// TIA Portal V17 export
// export: Created 2025-03-10T13:11:52.5932602Z, ExportSetting WithDefaults, DisplayName Totally Integrated Automation Portal, DisplayVersion V17 Update 8, DisplayName TIA Portal Openness, DisplayVersion V17 Update 8, DisplayName TIA Portal Version Control Interface, DisplayVersion V17, DisplayName SINAMICS Startdrive Advanced, DisplayVersion V17 SP2, DisplayName SINAMICS Startdrive G110M, G120, G120C, G120D, G120P, G115D, DisplayVersion V17 SP2, DisplayName SINAMICS Startdrive G130, G150, S120, S150, SINAMICS MV, S210, DisplayVersion V17 SP2, DisplayName STEP 7 Professional, DisplayVersion V17 Update 8, DisplayName SINUMERIK ONE STEP 7 Toolbox, DisplayVersion V17 Update 12, DisplayName SINUMERIK 840D sl STEP 7 Toolbox, DisplayVersion V17 Update 12, DisplayName STEP 7 Safety, DisplayVersion V17 Update 6, DisplayName WinCC Advanced, DisplayVersion V17 Update 8
TYPE "LBP_typeAlarmMsgs"
TITLE = PLC-Error / Messages / PLC errores/avisos / PLC-Fehler / Meldungen
// User data type for block LBP_AlarmMessage [DB2] / Tipo de dato de usuario para bloque LBP_AlarmMessage [DB2] / Anwender-Datentyp für Baustein LBP_AlarmMessage [DB2]
// stored: IsFailsafeCompliant false
   STRUCT
      Chan : Array[1..10] of Struct   // Von Kanal 1..10 / From Channel 1..10 / Desde el canal 1..10
         FDD : Array[0..15] of Bool;   // Vorschub deaktivieren / Feed disable / Desactivar avance
         RID : Array[0..15] of Bool;   // Einlesen deaktivieren / Read-in disable / Desactivar lectura
         NCSD : Array[0..15] of Bool;   // NC Start deaktivieren / NC start disable / Desactivar Marcha CN
         FdStop_1 : Array[0..15] of Bool;   // Vorschub-Stopp GEO-Achse 1 / Feed stop GEOaxis 1 / Parada del avance eje geométrico 1
         FdStop_2 : Array[0..15] of Bool;   // Vorschub-Stopp GEO-Achse 2 / Feed stop GEOaxis 2 / Parada del avance eje geométrico 2
         FdStop_3 : Array[0..15] of Bool;   // Vorschub-Stopp GEO-Achse 3 / Feed stop GEOaxis 3 / Parada del avance eje geométrico 3
      END_STRUCT;
      Axis : Array[1..31] of Struct   // Von Achse 1..31 / From Axis 1..31 / Desde el eje 1..31
         FdStop : Array[0..15] of Bool;   // Vorschub-Stopp Achse/Spindel / Feed stop axis/spindle / Parada del avance eje/cabezal
      END_STRUCT;
      AddValUserA0 : Array[0..63] of Int;   // Zusätzlicher Wert für Alarme im Anwenderbereich 0 (700000..700063) / Additional value for alarms in the user area 0 (700000..700063) / Valor adicional para alarmas en el área de usuario 0 (700000..700063)
      ChanA : Array[1..10] of Struct   // Von Kanal 1..10 / From Channel 1..10 / Desde el canal 1..10
         FDD_5C00xx : Array[0..15] of Bool;   // Vorschub deaktivieren Alarm Nr. 5C0000..5C0015 / Feed disable Alarm no. 5C0000..5C0015 / Desactivar avance n.º alarma 5C0000..5C0015
         FDD_RID_5C01xx : Array[0..31] of Bool;   // Vorschub und Einlesen deaktivieren Alarm Nr. 5C0100..5C0131 / Feed and read-in disable Alarm no. 5C0100..5C0131 / Desactivar avance y lectura n.º alarma 5C0100..5C0131
         RID_5C02xx : Array[0..31] of Bool;   // Einlesen deaktivieren Alarm Nr. 5C0200..5C0231 / Read-in disable Alarm no. 5C0200..5C0231 / Desactivar lectura n.º alarma 5C0200..5C0231
         NCSD_5C03xx : Array[0..15] of Bool;   // NC Start deaktivieren Alarm Nr. 5C0300..5C0315 / NC start disable Alarm no. 5C0300..5C0315 / Desactivar Marcha CN n.º alarma 5C0300..5C0315
         FdStop_1_5C11xx : Array[0..15] of Bool;   // Vorschub-Stopp GEO-Achse 1 Alarm Nr. 5C1100..5C1115 / Feed stop GEOaxis 1 Alarm no. 5C1100..5C1115 / Parada de avance eje geométrico 1 n.º alarma 5C1100..5C1115
         FdStop_2_5C12xx : Array[0..15] of Bool;   // Vorschub-Stopp GEO-Achse 2 Alarm Nr. 5C1200..5C1215 / Feed stop GEOaxis 2 Alarm no. 5C1200..5C1215 / Parada de avance eje geométrico 2 n.º alarma 5C1200..5C1215
         FdStop_3_5C13xx : Array[0..15] of Bool;   // Vorschub-Stopp GEO-Achse 3 Alarm Nr. 5C1300..5C1315 / Feed stop GEOaxis 3 Alarm no. 5C1300..5C1315 / Parada de avance eje geométrico 3 n.º alarma 5C1300..5C1315
      END_STRUCT;
      AxisA : Array[1..31] of Struct   // Von Achse 1..31 / From Axis 1..31 / Desde el eje 1..31
         AAFdStop60AAxx : Array[0..15] of Bool;   // Vorschub-Stopp Achse/Spindel / Feed stop axis/spindle / Parada del avance eje/cabezal
      END_STRUCT;
      res552 : Word;   // Reserviert / Reserved / Reservado
      UserA : Array[0..63] of Struct
         A70UUxx : Array[0..63] of Bool;   // Alarm 70UU00..70UU63 (Anwender-Bereich) / Alarm 70UU00..70UU63 (user area) / Alarma 70UU00..70UU63 (área de usuario)
      END_STRUCT;
   END_STRUCT;
   // // Chan[2].FDD : Vorschub deaktivieren / Feed disable / Desactivar avance
   // // Chan[3].FDD : Vorschub deaktivieren / Feed disable / Desactivar avance
   // // Chan[4].FDD : Vorschub deaktivieren / Feed disable / Desactivar avance
   // // Chan[5].FDD : Vorschub deaktivieren / Feed disable / Desactivar avance
   // // Chan[6].FDD : Vorschub deaktivieren / Feed disable / Desactivar avance
   // // Chan[7].FDD : Vorschub deaktivieren / Feed disable / Desactivar avance
   // // Chan[8].FDD : Vorschub deaktivieren / Feed disable / Desactivar avance
   // // Chan[9].FDD : Vorschub deaktivieren / Feed disable / Desactivar avance
   // // Chan[10].FDD : Vorschub deaktivieren / Feed disable / Desactivar avance
   // // Chan[2].RID : Einlesen deaktivieren / Read-in disable / Desactivar lectura
   // // Chan[3].RID : Einlesen deaktivieren / Read-in disable / Desactivar lectura
   // // Chan[4].RID : Einlesen deaktivieren / Read-in disable / Desactivar lectura
   // // Chan[5].RID : Einlesen deaktivieren / Read-in disable / Desactivar lectura
   // // Chan[6].RID : Einlesen deaktivieren / Read-in disable / Desactivar lectura
   // // Chan[7].RID : Einlesen deaktivieren / Read-in disable / Desactivar lectura
   // // Chan[8].RID : Einlesen deaktivieren / Read-in disable / Desactivar lectura
   // // Chan[9].RID : Einlesen deaktivieren / Read-in disable / Desactivar lectura
   // // Chan[10].RID : Einlesen deaktivieren / Read-in disable / Desactivar lectura
   // // Chan[2].NCSD : NC Start deaktivieren / NC start disable / Desactivar Marcha CN
   // // Chan[3].NCSD : NC Start deaktivieren / NC start disable / Desactivar Marcha CN
   // // Chan[4].NCSD : NC Start deaktivieren / NC start disable / Desactivar Marcha CN
   // // Chan[5].NCSD : NC Start deaktivieren / NC start disable / Desactivar Marcha CN
   // // Chan[6].NCSD : NC Start deaktivieren / NC start disable / Desactivar Marcha CN
   // // Chan[7].NCSD : NC Start deaktivieren / NC start disable / Desactivar Marcha CN
   // // Chan[8].NCSD : NC Start deaktivieren / NC start disable / Desactivar Marcha CN
   // // Chan[9].NCSD : NC Start deaktivieren / NC start disable / Desactivar Marcha CN
   // // Chan[10].NCSD : NC Start deaktivieren / NC start disable / Desactivar Marcha CN
   // // Chan[2].FdStop_1 : Vorschub-Stopp GEO-Achse 1 / Feed stop GEOaxis 1 / Parada del avance eje geométrico 1
   // // Chan[3].FdStop_1 : Vorschub-Stopp GEO-Achse 1 / Feed stop GEOaxis 1 / Parada del avance eje geométrico 1
   // // Chan[4].FdStop_1 : Vorschub-Stopp GEO-Achse 1 / Feed stop GEOaxis 1 / Parada del avance eje geométrico 1
   // // Chan[5].FdStop_1 : Vorschub-Stopp GEO-Achse 1 / Feed stop GEOaxis 1 / Parada del avance eje geométrico 1
   // // Chan[6].FdStop_1 : Vorschub-Stopp GEO-Achse 1 / Feed stop GEOaxis 1 / Parada del avance eje geométrico 1
   // // Chan[7].FdStop_1 : Vorschub-Stopp GEO-Achse 1 / Feed stop GEOaxis 1 / Parada del avance eje geométrico 1
   // // Chan[8].FdStop_1 : Vorschub-Stopp GEO-Achse 1 / Feed stop GEOaxis 1 / Parada del avance eje geométrico 1
   // // Chan[9].FdStop_1 : Vorschub-Stopp GEO-Achse 1 / Feed stop GEOaxis 1 / Parada del avance eje geométrico 1
   // // Chan[10].FdStop_1 : Vorschub-Stopp GEO-Achse 1 / Feed stop GEOaxis 1 / Parada del avance eje geométrico 1
   // // Chan[2].FdStop_2 : Vorschub-Stopp GEO-Achse 2 / Feed stop GEOaxis 2 / Parada del avance eje geométrico 2
   // // Chan[3].FdStop_2 : Vorschub-Stopp GEO-Achse 2 / Feed stop GEOaxis 2 / Parada del avance eje geométrico 2
   // // Chan[4].FdStop_2 : Vorschub-Stopp GEO-Achse 2 / Feed stop GEOaxis 2 / Parada del avance eje geométrico 2
   // // Chan[5].FdStop_2 : Vorschub-Stopp GEO-Achse 2 / Feed stop GEOaxis 2 / Parada del avance eje geométrico 2
   // // Chan[6].FdStop_2 : Vorschub-Stopp GEO-Achse 2 / Feed stop GEOaxis 2 / Parada del avance eje geométrico 2
   // // Chan[7].FdStop_2 : Vorschub-Stopp GEO-Achse 2 / Feed stop GEOaxis 2 / Parada del avance eje geométrico 2
   // // Chan[8].FdStop_2 : Vorschub-Stopp GEO-Achse 2 / Feed stop GEOaxis 2 / Parada del avance eje geométrico 2
   // // Chan[9].FdStop_2 : Vorschub-Stopp GEO-Achse 2 / Feed stop GEOaxis 2 / Parada del avance eje geométrico 2
   // // Chan[10].FdStop_2 : Vorschub-Stopp GEO-Achse 2 / Feed stop GEOaxis 2 / Parada del avance eje geométrico 2
   // // Chan[2].FdStop_3 : Vorschub-Stopp GEO-Achse 3 / Feed stop GEOaxis 3 / Parada del avance eje geométrico 3
   // // Chan[3].FdStop_3 : Vorschub-Stopp GEO-Achse 3 / Feed stop GEOaxis 3 / Parada del avance eje geométrico 3
   // // Chan[4].FdStop_3 : Vorschub-Stopp GEO-Achse 3 / Feed stop GEOaxis 3 / Parada del avance eje geométrico 3
   // // Chan[5].FdStop_3 : Vorschub-Stopp GEO-Achse 3 / Feed stop GEOaxis 3 / Parada del avance eje geométrico 3
   // // Chan[6].FdStop_3 : Vorschub-Stopp GEO-Achse 3 / Feed stop GEOaxis 3 / Parada del avance eje geométrico 3
   // // Chan[7].FdStop_3 : Vorschub-Stopp GEO-Achse 3 / Feed stop GEOaxis 3 / Parada del avance eje geométrico 3
   // // Chan[8].FdStop_3 : Vorschub-Stopp GEO-Achse 3 / Feed stop GEOaxis 3 / Parada del avance eje geométrico 3
   // // Chan[9].FdStop_3 : Vorschub-Stopp GEO-Achse 3 / Feed stop GEOaxis 3 / Parada del avance eje geométrico 3
   // // Chan[10].FdStop_3 : Vorschub-Stopp GEO-Achse 3 / Feed stop GEOaxis 3 / Parada del avance eje geométrico 3
   // // Chan[1] : Von Kanal 1..10 / From Channel 1..10 / Desde el canal 1..10
   // // Chan[2] : Von Kanal 1..10 / From Channel 1..10 / Desde el canal 1..10
   // // Chan[3] : Von Kanal 1..10 / From Channel 1..10 / Desde el canal 1..10
   // // Chan[4] : Von Kanal 1..10 / From Channel 1..10 / Desde el canal 1..10
   // // Chan[5] : Von Kanal 1..10 / From Channel 1..10 / Desde el canal 1..10
   // // Chan[6] : Von Kanal 1..10 / From Channel 1..10 / Desde el canal 1..10
   // // Chan[7] : Von Kanal 1..10 / From Channel 1..10 / Desde el canal 1..10
   // // Chan[8] : Von Kanal 1..10 / From Channel 1..10 / Desde el canal 1..10
   // // Chan[9] : Von Kanal 1..10 / From Channel 1..10 / Desde el canal 1..10
   // // Chan[10] : Von Kanal 1..10 / From Channel 1..10 / Desde el canal 1..10
   // // Axis[2].FdStop : Vorschub-Stopp Achse/Spindel / Feed stop axis/spindle / Parada del avance eje/cabezal
   // // Axis[3].FdStop : Vorschub-Stopp Achse/Spindel / Feed stop axis/spindle / Parada del avance eje/cabezal
   // // Axis[4].FdStop : Vorschub-Stopp Achse/Spindel / Feed stop axis/spindle / Parada del avance eje/cabezal
   // // Axis[5].FdStop : Vorschub-Stopp Achse/Spindel / Feed stop axis/spindle / Parada del avance eje/cabezal
   // // Axis[6].FdStop : Vorschub-Stopp Achse/Spindel / Feed stop axis/spindle / Parada del avance eje/cabezal
   // // Axis[7].FdStop : Vorschub-Stopp Achse/Spindel / Feed stop axis/spindle / Parada del avance eje/cabezal
   // // Axis[8].FdStop : Vorschub-Stopp Achse/Spindel / Feed stop axis/spindle / Parada del avance eje/cabezal
   // // Axis[9].FdStop : Vorschub-Stopp Achse/Spindel / Feed stop axis/spindle / Parada del avance eje/cabezal
   // // Axis[10].FdStop : Vorschub-Stopp Achse/Spindel / Feed stop axis/spindle / Parada del avance eje/cabezal
   // // Axis[11].FdStop : Vorschub-Stopp Achse/Spindel / Feed stop axis/spindle / Parada del avance eje/cabezal
   // // Axis[12].FdStop : Vorschub-Stopp Achse/Spindel / Feed stop axis/spindle / Parada del avance eje/cabezal
   // // Axis[13].FdStop : Vorschub-Stopp Achse/Spindel / Feed stop axis/spindle / Parada del avance eje/cabezal
   // // Axis[14].FdStop : Vorschub-Stopp Achse/Spindel / Feed stop axis/spindle / Parada del avance eje/cabezal
   // // Axis[15].FdStop : Vorschub-Stopp Achse/Spindel / Feed stop axis/spindle / Parada del avance eje/cabezal
   // // Axis[16].FdStop : Vorschub-Stopp Achse/Spindel / Feed stop axis/spindle / Parada del avance eje/cabezal
   // // Axis[17].FdStop : Vorschub-Stopp Achse/Spindel / Feed stop axis/spindle / Parada del avance eje/cabezal
   // // Axis[18].FdStop : Vorschub-Stopp Achse/Spindel / Feed stop axis/spindle / Parada del avance eje/cabezal
   // // Axis[19].FdStop : Vorschub-Stopp Achse/Spindel / Feed stop axis/spindle / Parada del avance eje/cabezal
   // // Axis[20].FdStop : Vorschub-Stopp Achse/Spindel / Feed stop axis/spindle / Parada del avance eje/cabezal
   // // Axis[21].FdStop : Vorschub-Stopp Achse/Spindel / Feed stop axis/spindle / Parada del avance eje/cabezal
   // // Axis[22].FdStop : Vorschub-Stopp Achse/Spindel / Feed stop axis/spindle / Parada del avance eje/cabezal
   // // Axis[23].FdStop : Vorschub-Stopp Achse/Spindel / Feed stop axis/spindle / Parada del avance eje/cabezal
   // // Axis[24].FdStop : Vorschub-Stopp Achse/Spindel / Feed stop axis/spindle / Parada del avance eje/cabezal
   // // Axis[25].FdStop : Vorschub-Stopp Achse/Spindel / Feed stop axis/spindle / Parada del avance eje/cabezal
   // // Axis[26].FdStop : Vorschub-Stopp Achse/Spindel / Feed stop axis/spindle / Parada del avance eje/cabezal
   // // Axis[27].FdStop : Vorschub-Stopp Achse/Spindel / Feed stop axis/spindle / Parada del avance eje/cabezal
   // // Axis[28].FdStop : Vorschub-Stopp Achse/Spindel / Feed stop axis/spindle / Parada del avance eje/cabezal
   // // Axis[29].FdStop : Vorschub-Stopp Achse/Spindel / Feed stop axis/spindle / Parada del avance eje/cabezal
   // // Axis[30].FdStop : Vorschub-Stopp Achse/Spindel / Feed stop axis/spindle / Parada del avance eje/cabezal
   // // Axis[31].FdStop : Vorschub-Stopp Achse/Spindel / Feed stop axis/spindle / Parada del avance eje/cabezal
   // // Axis[1] : Von Achse 1..31 / From Axis 1..31 / Desde el eje 1..31
   // // Axis[2] : Von Achse 1..31 / From Axis 1..31 / Desde el eje 1..31
   // // Axis[3] : Von Achse 1..31 / From Axis 1..31 / Desde el eje 1..31
   // // Axis[4] : Von Achse 1..31 / From Axis 1..31 / Desde el eje 1..31
   // // Axis[5] : Von Achse 1..31 / From Axis 1..31 / Desde el eje 1..31
   // // Axis[6] : Von Achse 1..31 / From Axis 1..31 / Desde el eje 1..31
   // // Axis[7] : Von Achse 1..31 / From Axis 1..31 / Desde el eje 1..31
   // // Axis[8] : Von Achse 1..31 / From Axis 1..31 / Desde el eje 1..31
   // // Axis[9] : Von Achse 1..31 / From Axis 1..31 / Desde el eje 1..31
   // // Axis[10] : Von Achse 1..31 / From Axis 1..31 / Desde el eje 1..31
   // // Axis[11] : Von Achse 1..31 / From Axis 1..31 / Desde el eje 1..31
   // // Axis[12] : Von Achse 1..31 / From Axis 1..31 / Desde el eje 1..31
   // // Axis[13] : Von Achse 1..31 / From Axis 1..31 / Desde el eje 1..31
   // // Axis[14] : Von Achse 1..31 / From Axis 1..31 / Desde el eje 1..31
   // // Axis[15] : Von Achse 1..31 / From Axis 1..31 / Desde el eje 1..31
   // // Axis[16] : Von Achse 1..31 / From Axis 1..31 / Desde el eje 1..31
   // // Axis[17] : Von Achse 1..31 / From Axis 1..31 / Desde el eje 1..31
   // // Axis[18] : Von Achse 1..31 / From Axis 1..31 / Desde el eje 1..31
   // // Axis[19] : Von Achse 1..31 / From Axis 1..31 / Desde el eje 1..31
   // // Axis[20] : Von Achse 1..31 / From Axis 1..31 / Desde el eje 1..31
   // // Axis[21] : Von Achse 1..31 / From Axis 1..31 / Desde el eje 1..31
   // // Axis[22] : Von Achse 1..31 / From Axis 1..31 / Desde el eje 1..31
   // // Axis[23] : Von Achse 1..31 / From Axis 1..31 / Desde el eje 1..31
   // // Axis[24] : Von Achse 1..31 / From Axis 1..31 / Desde el eje 1..31
   // // Axis[25] : Von Achse 1..31 / From Axis 1..31 / Desde el eje 1..31
   // // Axis[26] : Von Achse 1..31 / From Axis 1..31 / Desde el eje 1..31
   // // Axis[27] : Von Achse 1..31 / From Axis 1..31 / Desde el eje 1..31
   // // Axis[28] : Von Achse 1..31 / From Axis 1..31 / Desde el eje 1..31
   // // Axis[29] : Von Achse 1..31 / From Axis 1..31 / Desde el eje 1..31
   // // Axis[30] : Von Achse 1..31 / From Axis 1..31 / Desde el eje 1..31
   // // Axis[31] : Von Achse 1..31 / From Axis 1..31 / Desde el eje 1..31
   // // ChanA[2].FDD_5C00xx : Vorschub deaktivieren Alarm Nr. 5C0000..5C0015 / Feed disable Alarm no. 5C0000..5C0015 / Desactivar avance n.º alarma 5C0000..5C0015
   // // ChanA[3].FDD_5C00xx : Vorschub deaktivieren Alarm Nr. 5C0000..5C0015 / Feed disable Alarm no. 5C0000..5C0015 / Desactivar avance n.º alarma 5C0000..5C0015
   // // ChanA[4].FDD_5C00xx : Vorschub deaktivieren Alarm Nr. 5C0000..5C0015 / Feed disable Alarm no. 5C0000..5C0015 / Desactivar avance n.º alarma 5C0000..5C0015
   // // ChanA[5].FDD_5C00xx : Vorschub deaktivieren Alarm Nr. 5C0000..5C0015 / Feed disable Alarm no. 5C0000..5C0015 / Desactivar avance n.º alarma 5C0000..5C0015
   // // ChanA[6].FDD_5C00xx : Vorschub deaktivieren Alarm Nr. 5C0000..5C0015 / Feed disable Alarm no. 5C0000..5C0015 / Desactivar avance n.º alarma 5C0000..5C0015
   // // ChanA[7].FDD_5C00xx : Vorschub deaktivieren Alarm Nr. 5C0000..5C0015 / Feed disable Alarm no. 5C0000..5C0015 / Desactivar avance n.º alarma 5C0000..5C0015
   // // ChanA[8].FDD_5C00xx : Vorschub deaktivieren Alarm Nr. 5C0000..5C0015 / Feed disable Alarm no. 5C0000..5C0015 / Desactivar avance n.º alarma 5C0000..5C0015
   // // ChanA[9].FDD_5C00xx : Vorschub deaktivieren Alarm Nr. 5C0000..5C0015 / Feed disable Alarm no. 5C0000..5C0015 / Desactivar avance n.º alarma 5C0000..5C0015
   // // ChanA[10].FDD_5C00xx : Vorschub deaktivieren Alarm Nr. 5C0000..5C0015 / Feed disable Alarm no. 5C0000..5C0015 / Desactivar avance n.º alarma 5C0000..5C0015
   // // ChanA[2].FDD_RID_5C01xx : Vorschub und Einlesen deaktivieren Alarm Nr. 5C0100..5C0131 / Feed and read-in disable Alarm no. 5C0100..5C0131 / Desactivar avance y lectura n.º alarma 5C0100..5C0131
   // // ChanA[3].FDD_RID_5C01xx : Vorschub und Einlesen deaktivieren Alarm Nr. 5C0100..5C0131 / Feed and read-in disable Alarm no. 5C0100..5C0131 / Desactivar avance y lectura n.º alarma 5C0100..5C0131
   // // ChanA[4].FDD_RID_5C01xx : Vorschub und Einlesen deaktivieren Alarm Nr. 5C0100..5C0131 / Feed and read-in disable Alarm no. 5C0100..5C0131 / Desactivar avance y lectura n.º alarma 5C0100..5C0131
   // // ChanA[5].FDD_RID_5C01xx : Vorschub und Einlesen deaktivieren Alarm Nr. 5C0100..5C0131 / Feed and read-in disable Alarm no. 5C0100..5C0131 / Desactivar avance y lectura n.º alarma 5C0100..5C0131
   // // ChanA[6].FDD_RID_5C01xx : Vorschub und Einlesen deaktivieren Alarm Nr. 5C0100..5C0131 / Feed and read-in disable Alarm no. 5C0100..5C0131 / Desactivar avance y lectura n.º alarma 5C0100..5C0131
   // // ChanA[7].FDD_RID_5C01xx : Vorschub und Einlesen deaktivieren Alarm Nr. 5C0100..5C0131 / Feed and read-in disable Alarm no. 5C0100..5C0131 / Desactivar avance y lectura n.º alarma 5C0100..5C0131
   // // ChanA[8].FDD_RID_5C01xx : Vorschub und Einlesen deaktivieren Alarm Nr. 5C0100..5C0131 / Feed and read-in disable Alarm no. 5C0100..5C0131 / Desactivar avance y lectura n.º alarma 5C0100..5C0131
   // // ChanA[9].FDD_RID_5C01xx : Vorschub und Einlesen deaktivieren Alarm Nr. 5C0100..5C0131 / Feed and read-in disable Alarm no. 5C0100..5C0131 / Desactivar avance y lectura n.º alarma 5C0100..5C0131
   // // ChanA[10].FDD_RID_5C01xx : Vorschub und Einlesen deaktivieren Alarm Nr. 5C0100..5C0131 / Feed and read-in disable Alarm no. 5C0100..5C0131 / Desactivar avance y lectura n.º alarma 5C0100..5C0131
   // // ChanA[2].RID_5C02xx : Einlesen deaktivieren Alarm Nr. 5C0200..5C0231 / Read-in disable Alarm no. 5C0200..5C0231 / Desactivar lectura n.º alarma 5C0200..5C0231
   // // ChanA[3].RID_5C02xx : Einlesen deaktivieren Alarm Nr. 5C0200..5C0231 / Read-in disable Alarm no. 5C0200..5C0231 / Desactivar lectura n.º alarma 5C0200..5C0231
   // // ChanA[4].RID_5C02xx : Einlesen deaktivieren Alarm Nr. 5C0200..5C0231 / Read-in disable Alarm no. 5C0200..5C0231 / Desactivar lectura n.º alarma 5C0200..5C0231
   // // ChanA[5].RID_5C02xx : Einlesen deaktivieren Alarm Nr. 5C0200..5C0231 / Read-in disable Alarm no. 5C0200..5C0231 / Desactivar lectura n.º alarma 5C0200..5C0231
   // // ChanA[6].RID_5C02xx : Einlesen deaktivieren Alarm Nr. 5C0200..5C0231 / Read-in disable Alarm no. 5C0200..5C0231 / Desactivar lectura n.º alarma 5C0200..5C0231
   // // ChanA[7].RID_5C02xx : Einlesen deaktivieren Alarm Nr. 5C0200..5C0231 / Read-in disable Alarm no. 5C0200..5C0231 / Desactivar lectura n.º alarma 5C0200..5C0231
   // // ChanA[8].RID_5C02xx : Einlesen deaktivieren Alarm Nr. 5C0200..5C0231 / Read-in disable Alarm no. 5C0200..5C0231 / Desactivar lectura n.º alarma 5C0200..5C0231
   // // ChanA[9].RID_5C02xx : Einlesen deaktivieren Alarm Nr. 5C0200..5C0231 / Read-in disable Alarm no. 5C0200..5C0231 / Desactivar lectura n.º alarma 5C0200..5C0231
   // // ChanA[10].RID_5C02xx : Einlesen deaktivieren Alarm Nr. 5C0200..5C0231 / Read-in disable Alarm no. 5C0200..5C0231 / Desactivar lectura n.º alarma 5C0200..5C0231
   // // ChanA[2].NCSD_5C03xx : NC Start deaktivieren Alarm Nr. 5C0300..5C0315 / NC start disable Alarm no. 5C0300..5C0315 / Desactivar Marcha CN n.º alarma 5C0300..5C0315
   // // ChanA[3].NCSD_5C03xx : NC Start deaktivieren Alarm Nr. 5C0300..5C0315 / NC start disable Alarm no. 5C0300..5C0315 / Desactivar Marcha CN n.º alarma 5C0300..5C0315
   // // ChanA[4].NCSD_5C03xx : NC Start deaktivieren Alarm Nr. 5C0300..5C0315 / NC start disable Alarm no. 5C0300..5C0315 / Desactivar Marcha CN n.º alarma 5C0300..5C0315
   // // ChanA[5].NCSD_5C03xx : NC Start deaktivieren Alarm Nr. 5C0300..5C0315 / NC start disable Alarm no. 5C0300..5C0315 / Desactivar Marcha CN n.º alarma 5C0300..5C0315
   // // ChanA[6].NCSD_5C03xx : NC Start deaktivieren Alarm Nr. 5C0300..5C0315 / NC start disable Alarm no. 5C0300..5C0315 / Desactivar Marcha CN n.º alarma 5C0300..5C0315
   // // ChanA[7].NCSD_5C03xx : NC Start deaktivieren Alarm Nr. 5C0300..5C0315 / NC start disable Alarm no. 5C0300..5C0315 / Desactivar Marcha CN n.º alarma 5C0300..5C0315
   // // ChanA[8].NCSD_5C03xx : NC Start deaktivieren Alarm Nr. 5C0300..5C0315 / NC start disable Alarm no. 5C0300..5C0315 / Desactivar Marcha CN n.º alarma 5C0300..5C0315
   // // ChanA[9].NCSD_5C03xx : NC Start deaktivieren Alarm Nr. 5C0300..5C0315 / NC start disable Alarm no. 5C0300..5C0315 / Desactivar Marcha CN n.º alarma 5C0300..5C0315
   // // ChanA[10].NCSD_5C03xx : NC Start deaktivieren Alarm Nr. 5C0300..5C0315 / NC start disable Alarm no. 5C0300..5C0315 / Desactivar Marcha CN n.º alarma 5C0300..5C0315
   // // ChanA[2].FdStop_1_5C11xx : Vorschub-Stopp GEO-Achse 1 Alarm Nr. 5C1100..5C1115 / Feed stop GEOaxis 1 Alarm no. 5C1100..5C1115 / Parada de avance eje geométrico 1 n.º alarma 5C1100..5C1115
   // // ChanA[3].FdStop_1_5C11xx : Vorschub-Stopp GEO-Achse 1 Alarm Nr. 5C1100..5C1115 / Feed stop GEOaxis 1 Alarm no. 5C1100..5C1115 / Parada de avance eje geométrico 1 n.º alarma 5C1100..5C1115
   // // ChanA[4].FdStop_1_5C11xx : Vorschub-Stopp GEO-Achse 1 Alarm Nr. 5C1100..5C1115 / Feed stop GEOaxis 1 Alarm no. 5C1100..5C1115 / Parada de avance eje geométrico 1 n.º alarma 5C1100..5C1115
   // // ChanA[5].FdStop_1_5C11xx : Vorschub-Stopp GEO-Achse 1 Alarm Nr. 5C1100..5C1115 / Feed stop GEOaxis 1 Alarm no. 5C1100..5C1115 / Parada de avance eje geométrico 1 n.º alarma 5C1100..5C1115
   // // ChanA[6].FdStop_1_5C11xx : Vorschub-Stopp GEO-Achse 1 Alarm Nr. 5C1100..5C1115 / Feed stop GEOaxis 1 Alarm no. 5C1100..5C1115 / Parada de avance eje geométrico 1 n.º alarma 5C1100..5C1115
   // // ChanA[7].FdStop_1_5C11xx : Vorschub-Stopp GEO-Achse 1 Alarm Nr. 5C1100..5C1115 / Feed stop GEOaxis 1 Alarm no. 5C1100..5C1115 / Parada de avance eje geométrico 1 n.º alarma 5C1100..5C1115
   // // ChanA[8].FdStop_1_5C11xx : Vorschub-Stopp GEO-Achse 1 Alarm Nr. 5C1100..5C1115 / Feed stop GEOaxis 1 Alarm no. 5C1100..5C1115 / Parada de avance eje geométrico 1 n.º alarma 5C1100..5C1115
   // // ChanA[9].FdStop_1_5C11xx : Vorschub-Stopp GEO-Achse 1 Alarm Nr. 5C1100..5C1115 / Feed stop GEOaxis 1 Alarm no. 5C1100..5C1115 / Parada de avance eje geométrico 1 n.º alarma 5C1100..5C1115
   // // ChanA[10].FdStop_1_5C11xx : Vorschub-Stopp GEO-Achse 1 Alarm Nr. 5C1100..5C1115 / Feed stop GEOaxis 1 Alarm no. 5C1100..5C1115 / Parada de avance eje geométrico 1 n.º alarma 5C1100..5C1115
   // // ChanA[2].FdStop_2_5C12xx : Vorschub-Stopp GEO-Achse 2 Alarm Nr. 5C1200..5C1215 / Feed stop GEOaxis 2 Alarm no. 5C1200..5C1215 / Parada de avance eje geométrico 2 n.º alarma 5C1200..5C1215
   // // ChanA[3].FdStop_2_5C12xx : Vorschub-Stopp GEO-Achse 2 Alarm Nr. 5C1200..5C1215 / Feed stop GEOaxis 2 Alarm no. 5C1200..5C1215 / Parada de avance eje geométrico 2 n.º alarma 5C1200..5C1215
   // // ChanA[4].FdStop_2_5C12xx : Vorschub-Stopp GEO-Achse 2 Alarm Nr. 5C1200..5C1215 / Feed stop GEOaxis 2 Alarm no. 5C1200..5C1215 / Parada de avance eje geométrico 2 n.º alarma 5C1200..5C1215
   // // ChanA[5].FdStop_2_5C12xx : Vorschub-Stopp GEO-Achse 2 Alarm Nr. 5C1200..5C1215 / Feed stop GEOaxis 2 Alarm no. 5C1200..5C1215 / Parada de avance eje geométrico 2 n.º alarma 5C1200..5C1215
   // // ChanA[6].FdStop_2_5C12xx : Vorschub-Stopp GEO-Achse 2 Alarm Nr. 5C1200..5C1215 / Feed stop GEOaxis 2 Alarm no. 5C1200..5C1215 / Parada de avance eje geométrico 2 n.º alarma 5C1200..5C1215
   // // ChanA[7].FdStop_2_5C12xx : Vorschub-Stopp GEO-Achse 2 Alarm Nr. 5C1200..5C1215 / Feed stop GEOaxis 2 Alarm no. 5C1200..5C1215 / Parada de avance eje geométrico 2 n.º alarma 5C1200..5C1215
   // // ChanA[8].FdStop_2_5C12xx : Vorschub-Stopp GEO-Achse 2 Alarm Nr. 5C1200..5C1215 / Feed stop GEOaxis 2 Alarm no. 5C1200..5C1215 / Parada de avance eje geométrico 2 n.º alarma 5C1200..5C1215
   // // ChanA[9].FdStop_2_5C12xx : Vorschub-Stopp GEO-Achse 2 Alarm Nr. 5C1200..5C1215 / Feed stop GEOaxis 2 Alarm no. 5C1200..5C1215 / Parada de avance eje geométrico 2 n.º alarma 5C1200..5C1215
   // // ChanA[10].FdStop_2_5C12xx : Vorschub-Stopp GEO-Achse 2 Alarm Nr. 5C1200..5C1215 / Feed stop GEOaxis 2 Alarm no. 5C1200..5C1215 / Parada de avance eje geométrico 2 n.º alarma 5C1200..5C1215
   // // ChanA[2].FdStop_3_5C13xx : Vorschub-Stopp GEO-Achse 3 Alarm Nr. 5C1300..5C1315 / Feed stop GEOaxis 3 Alarm no. 5C1300..5C1315 / Parada de avance eje geométrico 3 n.º alarma 5C1300..5C1315
   // // ChanA[3].FdStop_3_5C13xx : Vorschub-Stopp GEO-Achse 3 Alarm Nr. 5C1300..5C1315 / Feed stop GEOaxis 3 Alarm no. 5C1300..5C1315 / Parada de avance eje geométrico 3 n.º alarma 5C1300..5C1315
   // // ChanA[4].FdStop_3_5C13xx : Vorschub-Stopp GEO-Achse 3 Alarm Nr. 5C1300..5C1315 / Feed stop GEOaxis 3 Alarm no. 5C1300..5C1315 / Parada de avance eje geométrico 3 n.º alarma 5C1300..5C1315
   // // ChanA[5].FdStop_3_5C13xx : Vorschub-Stopp GEO-Achse 3 Alarm Nr. 5C1300..5C1315 / Feed stop GEOaxis 3 Alarm no. 5C1300..5C1315 / Parada de avance eje geométrico 3 n.º alarma 5C1300..5C1315
   // // ChanA[6].FdStop_3_5C13xx : Vorschub-Stopp GEO-Achse 3 Alarm Nr. 5C1300..5C1315 / Feed stop GEOaxis 3 Alarm no. 5C1300..5C1315 / Parada de avance eje geométrico 3 n.º alarma 5C1300..5C1315
   // // ChanA[7].FdStop_3_5C13xx : Vorschub-Stopp GEO-Achse 3 Alarm Nr. 5C1300..5C1315 / Feed stop GEOaxis 3 Alarm no. 5C1300..5C1315 / Parada de avance eje geométrico 3 n.º alarma 5C1300..5C1315
   // // ChanA[8].FdStop_3_5C13xx : Vorschub-Stopp GEO-Achse 3 Alarm Nr. 5C1300..5C1315 / Feed stop GEOaxis 3 Alarm no. 5C1300..5C1315 / Parada de avance eje geométrico 3 n.º alarma 5C1300..5C1315
   // // ChanA[9].FdStop_3_5C13xx : Vorschub-Stopp GEO-Achse 3 Alarm Nr. 5C1300..5C1315 / Feed stop GEOaxis 3 Alarm no. 5C1300..5C1315 / Parada de avance eje geométrico 3 n.º alarma 5C1300..5C1315
   // // ChanA[10].FdStop_3_5C13xx : Vorschub-Stopp GEO-Achse 3 Alarm Nr. 5C1300..5C1315 / Feed stop GEOaxis 3 Alarm no. 5C1300..5C1315 / Parada de avance eje geométrico 3 n.º alarma 5C1300..5C1315
   // // ChanA[1] : Von Kanal 1..10 / From Channel 1..10 / Desde el canal 1..10
   // // ChanA[2] : Von Kanal 1..10 / From Channel 1..10 / Desde el canal 1..10
   // // ChanA[3] : Von Kanal 1..10 / From Channel 1..10 / Desde el canal 1..10
   // // ChanA[4] : Von Kanal 1..10 / From Channel 1..10 / Desde el canal 1..10
   // // ChanA[5] : Von Kanal 1..10 / From Channel 1..10 / Desde el canal 1..10
   // // ChanA[6] : Von Kanal 1..10 / From Channel 1..10 / Desde el canal 1..10
   // // ChanA[7] : Von Kanal 1..10 / From Channel 1..10 / Desde el canal 1..10
   // // ChanA[8] : Von Kanal 1..10 / From Channel 1..10 / Desde el canal 1..10
   // // ChanA[9] : Von Kanal 1..10 / From Channel 1..10 / Desde el canal 1..10
   // // ChanA[10] : Von Kanal 1..10 / From Channel 1..10 / Desde el canal 1..10
   // // AxisA[2].AAFdStop60AAxx : Vorschub-Stopp Achse/Spindel / Feed stop axis/spindle / Parada del avance eje/cabezal
   // // AxisA[3].AAFdStop60AAxx : Vorschub-Stopp Achse/Spindel / Feed stop axis/spindle / Parada del avance eje/cabezal
   // // AxisA[4].AAFdStop60AAxx : Vorschub-Stopp Achse/Spindel / Feed stop axis/spindle / Parada del avance eje/cabezal
   // // AxisA[5].AAFdStop60AAxx : Vorschub-Stopp Achse/Spindel / Feed stop axis/spindle / Parada del avance eje/cabezal
   // // AxisA[6].AAFdStop60AAxx : Vorschub-Stopp Achse/Spindel / Feed stop axis/spindle / Parada del avance eje/cabezal
   // // AxisA[7].AAFdStop60AAxx : Vorschub-Stopp Achse/Spindel / Feed stop axis/spindle / Parada del avance eje/cabezal
   // // AxisA[8].AAFdStop60AAxx : Vorschub-Stopp Achse/Spindel / Feed stop axis/spindle / Parada del avance eje/cabezal
   // // AxisA[9].AAFdStop60AAxx : Vorschub-Stopp Achse/Spindel / Feed stop axis/spindle / Parada del avance eje/cabezal
   // // AxisA[10].AAFdStop60AAxx : Vorschub-Stopp Achse/Spindel / Feed stop axis/spindle / Parada del avance eje/cabezal
   // // AxisA[11].AAFdStop60AAxx : Vorschub-Stopp Achse/Spindel / Feed stop axis/spindle / Parada del avance eje/cabezal
   // // AxisA[12].AAFdStop60AAxx : Vorschub-Stopp Achse/Spindel / Feed stop axis/spindle / Parada del avance eje/cabezal
   // // AxisA[13].AAFdStop60AAxx : Vorschub-Stopp Achse/Spindel / Feed stop axis/spindle / Parada del avance eje/cabezal
   // // AxisA[14].AAFdStop60AAxx : Vorschub-Stopp Achse/Spindel / Feed stop axis/spindle / Parada del avance eje/cabezal
   // // AxisA[15].AAFdStop60AAxx : Vorschub-Stopp Achse/Spindel / Feed stop axis/spindle / Parada del avance eje/cabezal
   // // AxisA[16].AAFdStop60AAxx : Vorschub-Stopp Achse/Spindel / Feed stop axis/spindle / Parada del avance eje/cabezal
   // // AxisA[17].AAFdStop60AAxx : Vorschub-Stopp Achse/Spindel / Feed stop axis/spindle / Parada del avance eje/cabezal
   // // AxisA[18].AAFdStop60AAxx : Vorschub-Stopp Achse/Spindel / Feed stop axis/spindle / Parada del avance eje/cabezal
   // // AxisA[19].AAFdStop60AAxx : Vorschub-Stopp Achse/Spindel / Feed stop axis/spindle / Parada del avance eje/cabezal
   // // AxisA[20].AAFdStop60AAxx : Vorschub-Stopp Achse/Spindel / Feed stop axis/spindle / Parada del avance eje/cabezal
   // // AxisA[21].AAFdStop60AAxx : Vorschub-Stopp Achse/Spindel / Feed stop axis/spindle / Parada del avance eje/cabezal
   // // AxisA[22].AAFdStop60AAxx : Vorschub-Stopp Achse/Spindel / Feed stop axis/spindle / Parada del avance eje/cabezal
   // // AxisA[23].AAFdStop60AAxx : Vorschub-Stopp Achse/Spindel / Feed stop axis/spindle / Parada del avance eje/cabezal
   // // AxisA[24].AAFdStop60AAxx : Vorschub-Stopp Achse/Spindel / Feed stop axis/spindle / Parada del avance eje/cabezal
   // // AxisA[25].AAFdStop60AAxx : Vorschub-Stopp Achse/Spindel / Feed stop axis/spindle / Parada del avance eje/cabezal
   // // AxisA[26].AAFdStop60AAxx : Vorschub-Stopp Achse/Spindel / Feed stop axis/spindle / Parada del avance eje/cabezal
   // // AxisA[27].AAFdStop60AAxx : Vorschub-Stopp Achse/Spindel / Feed stop axis/spindle / Parada del avance eje/cabezal
   // // AxisA[28].AAFdStop60AAxx : Vorschub-Stopp Achse/Spindel / Feed stop axis/spindle / Parada del avance eje/cabezal
   // // AxisA[29].AAFdStop60AAxx : Vorschub-Stopp Achse/Spindel / Feed stop axis/spindle / Parada del avance eje/cabezal
   // // AxisA[30].AAFdStop60AAxx : Vorschub-Stopp Achse/Spindel / Feed stop axis/spindle / Parada del avance eje/cabezal
   // // AxisA[31].AAFdStop60AAxx : Vorschub-Stopp Achse/Spindel / Feed stop axis/spindle / Parada del avance eje/cabezal
   // // AxisA[1] : Von Achse 1..31 / From Axis 1..31 / Desde el eje 1..31
   // // AxisA[2] : Von Achse 1..31 / From Axis 1..31 / Desde el eje 1..31
   // // AxisA[3] : Von Achse 1..31 / From Axis 1..31 / Desde el eje 1..31
   // // AxisA[4] : Von Achse 1..31 / From Axis 1..31 / Desde el eje 1..31
   // // AxisA[5] : Von Achse 1..31 / From Axis 1..31 / Desde el eje 1..31
   // // AxisA[6] : Von Achse 1..31 / From Axis 1..31 / Desde el eje 1..31
   // // AxisA[7] : Von Achse 1..31 / From Axis 1..31 / Desde el eje 1..31
   // // AxisA[8] : Von Achse 1..31 / From Axis 1..31 / Desde el eje 1..31
   // // AxisA[9] : Von Achse 1..31 / From Axis 1..31 / Desde el eje 1..31
   // // AxisA[10] : Von Achse 1..31 / From Axis 1..31 / Desde el eje 1..31
   // // AxisA[11] : Von Achse 1..31 / From Axis 1..31 / Desde el eje 1..31
   // // AxisA[12] : Von Achse 1..31 / From Axis 1..31 / Desde el eje 1..31
   // // AxisA[13] : Von Achse 1..31 / From Axis 1..31 / Desde el eje 1..31
   // // AxisA[14] : Von Achse 1..31 / From Axis 1..31 / Desde el eje 1..31
   // // AxisA[15] : Von Achse 1..31 / From Axis 1..31 / Desde el eje 1..31
   // // AxisA[16] : Von Achse 1..31 / From Axis 1..31 / Desde el eje 1..31
   // // AxisA[17] : Von Achse 1..31 / From Axis 1..31 / Desde el eje 1..31
   // // AxisA[18] : Von Achse 1..31 / From Axis 1..31 / Desde el eje 1..31
   // // AxisA[19] : Von Achse 1..31 / From Axis 1..31 / Desde el eje 1..31
   // // AxisA[20] : Von Achse 1..31 / From Axis 1..31 / Desde el eje 1..31
   // // AxisA[21] : Von Achse 1..31 / From Axis 1..31 / Desde el eje 1..31
   // // AxisA[22] : Von Achse 1..31 / From Axis 1..31 / Desde el eje 1..31
   // // AxisA[23] : Von Achse 1..31 / From Axis 1..31 / Desde el eje 1..31
   // // AxisA[24] : Von Achse 1..31 / From Axis 1..31 / Desde el eje 1..31
   // // AxisA[25] : Von Achse 1..31 / From Axis 1..31 / Desde el eje 1..31
   // // AxisA[26] : Von Achse 1..31 / From Axis 1..31 / Desde el eje 1..31
   // // AxisA[27] : Von Achse 1..31 / From Axis 1..31 / Desde el eje 1..31
   // // AxisA[28] : Von Achse 1..31 / From Axis 1..31 / Desde el eje 1..31
   // // AxisA[29] : Von Achse 1..31 / From Axis 1..31 / Desde el eje 1..31
   // // AxisA[30] : Von Achse 1..31 / From Axis 1..31 / Desde el eje 1..31
   // // AxisA[31] : Von Achse 1..31 / From Axis 1..31 / Desde el eje 1..31
   // // UserA[1].A70UUxx : Alarm 70UU00..70UU63 (Anwender-Bereich) / Alarm 70UU00..70UU63 (user area) / Alarma 70UU00..70UU63 (área de usuario)
   // // UserA[2].A70UUxx : Alarm 70UU00..70UU63 (Anwender-Bereich) / Alarm 70UU00..70UU63 (user area) / Alarma 70UU00..70UU63 (área de usuario)
   // // UserA[3].A70UUxx : Alarm 70UU00..70UU63 (Anwender-Bereich) / Alarm 70UU00..70UU63 (user area) / Alarma 70UU00..70UU63 (área de usuario)
   // // UserA[4].A70UUxx : Alarm 70UU00..70UU63 (Anwender-Bereich) / Alarm 70UU00..70UU63 (user area) / Alarma 70UU00..70UU63 (área de usuario)
   // // UserA[5].A70UUxx : Alarm 70UU00..70UU63 (Anwender-Bereich) / Alarm 70UU00..70UU63 (user area) / Alarma 70UU00..70UU63 (área de usuario)
   // // UserA[6].A70UUxx : Alarm 70UU00..70UU63 (Anwender-Bereich) / Alarm 70UU00..70UU63 (user area) / Alarma 70UU00..70UU63 (área de usuario)
   // // UserA[7].A70UUxx : Alarm 70UU00..70UU63 (Anwender-Bereich) / Alarm 70UU00..70UU63 (user area) / Alarma 70UU00..70UU63 (área de usuario)
   // // UserA[8].A70UUxx : Alarm 70UU00..70UU63 (Anwender-Bereich) / Alarm 70UU00..70UU63 (user area) / Alarma 70UU00..70UU63 (área de usuario)
   // // UserA[9].A70UUxx : Alarm 70UU00..70UU63 (Anwender-Bereich) / Alarm 70UU00..70UU63 (user area) / Alarma 70UU00..70UU63 (área de usuario)
   // // UserA[10].A70UUxx : Alarm 70UU00..70UU63 (Anwender-Bereich) / Alarm 70UU00..70UU63 (user area) / Alarma 70UU00..70UU63 (área de usuario)
   // // UserA[11].A70UUxx : Alarm 70UU00..70UU63 (Anwender-Bereich) / Alarm 70UU00..70UU63 (user area) / Alarma 70UU00..70UU63 (área de usuario)
   // // UserA[12].A70UUxx : Alarm 70UU00..70UU63 (Anwender-Bereich) / Alarm 70UU00..70UU63 (user area) / Alarma 70UU00..70UU63 (área de usuario)
   // // UserA[13].A70UUxx : Alarm 70UU00..70UU63 (Anwender-Bereich) / Alarm 70UU00..70UU63 (user area) / Alarma 70UU00..70UU63 (área de usuario)
   // // UserA[14].A70UUxx : Alarm 70UU00..70UU63 (Anwender-Bereich) / Alarm 70UU00..70UU63 (user area) / Alarma 70UU00..70UU63 (área de usuario)
   // // UserA[15].A70UUxx : Alarm 70UU00..70UU63 (Anwender-Bereich) / Alarm 70UU00..70UU63 (user area) / Alarma 70UU00..70UU63 (área de usuario)
   // // UserA[16].A70UUxx : Alarm 70UU00..70UU63 (Anwender-Bereich) / Alarm 70UU00..70UU63 (user area) / Alarma 70UU00..70UU63 (área de usuario)
   // // UserA[17].A70UUxx : Alarm 70UU00..70UU63 (Anwender-Bereich) / Alarm 70UU00..70UU63 (user area) / Alarma 70UU00..70UU63 (área de usuario)
   // // UserA[18].A70UUxx : Alarm 70UU00..70UU63 (Anwender-Bereich) / Alarm 70UU00..70UU63 (user area) / Alarma 70UU00..70UU63 (área de usuario)
   // // UserA[19].A70UUxx : Alarm 70UU00..70UU63 (Anwender-Bereich) / Alarm 70UU00..70UU63 (user area) / Alarma 70UU00..70UU63 (área de usuario)
   // // UserA[20].A70UUxx : Alarm 70UU00..70UU63 (Anwender-Bereich) / Alarm 70UU00..70UU63 (user area) / Alarma 70UU00..70UU63 (área de usuario)
   // // UserA[21].A70UUxx : Alarm 70UU00..70UU63 (Anwender-Bereich) / Alarm 70UU00..70UU63 (user area) / Alarma 70UU00..70UU63 (área de usuario)
   // // UserA[22].A70UUxx : Alarm 70UU00..70UU63 (Anwender-Bereich) / Alarm 70UU00..70UU63 (user area) / Alarma 70UU00..70UU63 (área de usuario)
   // // UserA[23].A70UUxx : Alarm 70UU00..70UU63 (Anwender-Bereich) / Alarm 70UU00..70UU63 (user area) / Alarma 70UU00..70UU63 (área de usuario)
   // // UserA[24].A70UUxx : Alarm 70UU00..70UU63 (Anwender-Bereich) / Alarm 70UU00..70UU63 (user area) / Alarma 70UU00..70UU63 (área de usuario)
   // // UserA[25].A70UUxx : Alarm 70UU00..70UU63 (Anwender-Bereich) / Alarm 70UU00..70UU63 (user area) / Alarma 70UU00..70UU63 (área de usuario)
   // // UserA[26].A70UUxx : Alarm 70UU00..70UU63 (Anwender-Bereich) / Alarm 70UU00..70UU63 (user area) / Alarma 70UU00..70UU63 (área de usuario)
   // // UserA[27].A70UUxx : Alarm 70UU00..70UU63 (Anwender-Bereich) / Alarm 70UU00..70UU63 (user area) / Alarma 70UU00..70UU63 (área de usuario)
   // // UserA[28].A70UUxx : Alarm 70UU00..70UU63 (Anwender-Bereich) / Alarm 70UU00..70UU63 (user area) / Alarma 70UU00..70UU63 (área de usuario)
   // // UserA[29].A70UUxx : Alarm 70UU00..70UU63 (Anwender-Bereich) / Alarm 70UU00..70UU63 (user area) / Alarma 70UU00..70UU63 (área de usuario)
   // // UserA[30].A70UUxx : Alarm 70UU00..70UU63 (Anwender-Bereich) / Alarm 70UU00..70UU63 (user area) / Alarma 70UU00..70UU63 (área de usuario)
   // // UserA[31].A70UUxx : Alarm 70UU00..70UU63 (Anwender-Bereich) / Alarm 70UU00..70UU63 (user area) / Alarma 70UU00..70UU63 (área de usuario)
   // // UserA[32].A70UUxx : Alarm 70UU00..70UU63 (Anwender-Bereich) / Alarm 70UU00..70UU63 (user area) / Alarma 70UU00..70UU63 (área de usuario)
   // // UserA[33].A70UUxx : Alarm 70UU00..70UU63 (Anwender-Bereich) / Alarm 70UU00..70UU63 (user area) / Alarma 70UU00..70UU63 (área de usuario)
   // // UserA[34].A70UUxx : Alarm 70UU00..70UU63 (Anwender-Bereich) / Alarm 70UU00..70UU63 (user area) / Alarma 70UU00..70UU63 (área de usuario)
   // // UserA[35].A70UUxx : Alarm 70UU00..70UU63 (Anwender-Bereich) / Alarm 70UU00..70UU63 (user area) / Alarma 70UU00..70UU63 (área de usuario)
   // // UserA[36].A70UUxx : Alarm 70UU00..70UU63 (Anwender-Bereich) / Alarm 70UU00..70UU63 (user area) / Alarma 70UU00..70UU63 (área de usuario)
   // // UserA[37].A70UUxx : Alarm 70UU00..70UU63 (Anwender-Bereich) / Alarm 70UU00..70UU63 (user area) / Alarma 70UU00..70UU63 (área de usuario)
   // // UserA[38].A70UUxx : Alarm 70UU00..70UU63 (Anwender-Bereich) / Alarm 70UU00..70UU63 (user area) / Alarma 70UU00..70UU63 (área de usuario)
   // // UserA[39].A70UUxx : Alarm 70UU00..70UU63 (Anwender-Bereich) / Alarm 70UU00..70UU63 (user area) / Alarma 70UU00..70UU63 (área de usuario)
   // // UserA[40].A70UUxx : Alarm 70UU00..70UU63 (Anwender-Bereich) / Alarm 70UU00..70UU63 (user area) / Alarma 70UU00..70UU63 (área de usuario)
   // // UserA[41].A70UUxx : Alarm 70UU00..70UU63 (Anwender-Bereich) / Alarm 70UU00..70UU63 (user area) / Alarma 70UU00..70UU63 (área de usuario)
   // // UserA[42].A70UUxx : Alarm 70UU00..70UU63 (Anwender-Bereich) / Alarm 70UU00..70UU63 (user area) / Alarma 70UU00..70UU63 (área de usuario)
   // // UserA[43].A70UUxx : Alarm 70UU00..70UU63 (Anwender-Bereich) / Alarm 70UU00..70UU63 (user area) / Alarma 70UU00..70UU63 (área de usuario)
   // // UserA[44].A70UUxx : Alarm 70UU00..70UU63 (Anwender-Bereich) / Alarm 70UU00..70UU63 (user area) / Alarma 70UU00..70UU63 (área de usuario)
   // // UserA[45].A70UUxx : Alarm 70UU00..70UU63 (Anwender-Bereich) / Alarm 70UU00..70UU63 (user area) / Alarma 70UU00..70UU63 (área de usuario)
   // // UserA[46].A70UUxx : Alarm 70UU00..70UU63 (Anwender-Bereich) / Alarm 70UU00..70UU63 (user area) / Alarma 70UU00..70UU63 (área de usuario)
   // // UserA[47].A70UUxx : Alarm 70UU00..70UU63 (Anwender-Bereich) / Alarm 70UU00..70UU63 (user area) / Alarma 70UU00..70UU63 (área de usuario)
   // // UserA[48].A70UUxx : Alarm 70UU00..70UU63 (Anwender-Bereich) / Alarm 70UU00..70UU63 (user area) / Alarma 70UU00..70UU63 (área de usuario)
   // // UserA[49].A70UUxx : Alarm 70UU00..70UU63 (Anwender-Bereich) / Alarm 70UU00..70UU63 (user area) / Alarma 70UU00..70UU63 (área de usuario)
   // // UserA[50].A70UUxx : Alarm 70UU00..70UU63 (Anwender-Bereich) / Alarm 70UU00..70UU63 (user area) / Alarma 70UU00..70UU63 (área de usuario)
   // // UserA[51].A70UUxx : Alarm 70UU00..70UU63 (Anwender-Bereich) / Alarm 70UU00..70UU63 (user area) / Alarma 70UU00..70UU63 (área de usuario)
   // // UserA[52].A70UUxx : Alarm 70UU00..70UU63 (Anwender-Bereich) / Alarm 70UU00..70UU63 (user area) / Alarma 70UU00..70UU63 (área de usuario)
   // // UserA[53].A70UUxx : Alarm 70UU00..70UU63 (Anwender-Bereich) / Alarm 70UU00..70UU63 (user area) / Alarma 70UU00..70UU63 (área de usuario)
   // // UserA[54].A70UUxx : Alarm 70UU00..70UU63 (Anwender-Bereich) / Alarm 70UU00..70UU63 (user area) / Alarma 70UU00..70UU63 (área de usuario)
   // // UserA[55].A70UUxx : Alarm 70UU00..70UU63 (Anwender-Bereich) / Alarm 70UU00..70UU63 (user area) / Alarma 70UU00..70UU63 (área de usuario)
   // // UserA[56].A70UUxx : Alarm 70UU00..70UU63 (Anwender-Bereich) / Alarm 70UU00..70UU63 (user area) / Alarma 70UU00..70UU63 (área de usuario)
   // // UserA[57].A70UUxx : Alarm 70UU00..70UU63 (Anwender-Bereich) / Alarm 70UU00..70UU63 (user area) / Alarma 70UU00..70UU63 (área de usuario)
   // // UserA[58].A70UUxx : Alarm 70UU00..70UU63 (Anwender-Bereich) / Alarm 70UU00..70UU63 (user area) / Alarma 70UU00..70UU63 (área de usuario)
   // // UserA[59].A70UUxx : Alarm 70UU00..70UU63 (Anwender-Bereich) / Alarm 70UU00..70UU63 (user area) / Alarma 70UU00..70UU63 (área de usuario)
   // // UserA[60].A70UUxx : Alarm 70UU00..70UU63 (Anwender-Bereich) / Alarm 70UU00..70UU63 (user area) / Alarma 70UU00..70UU63 (área de usuario)
   // // UserA[61].A70UUxx : Alarm 70UU00..70UU63 (Anwender-Bereich) / Alarm 70UU00..70UU63 (user area) / Alarma 70UU00..70UU63 (área de usuario)
   // // UserA[62].A70UUxx : Alarm 70UU00..70UU63 (Anwender-Bereich) / Alarm 70UU00..70UU63 (user area) / Alarma 70UU00..70UU63 (área de usuario)
   // // UserA[63].A70UUxx : Alarm 70UU00..70UU63 (Anwender-Bereich) / Alarm 70UU00..70UU63 (user area) / Alarma 70UU00..70UU63 (área de usuario)
END_TYPE
